// Mitsubishi GX Works2 project: 15속도제어   PLC: Q03UDV

PROGRAM MAIN
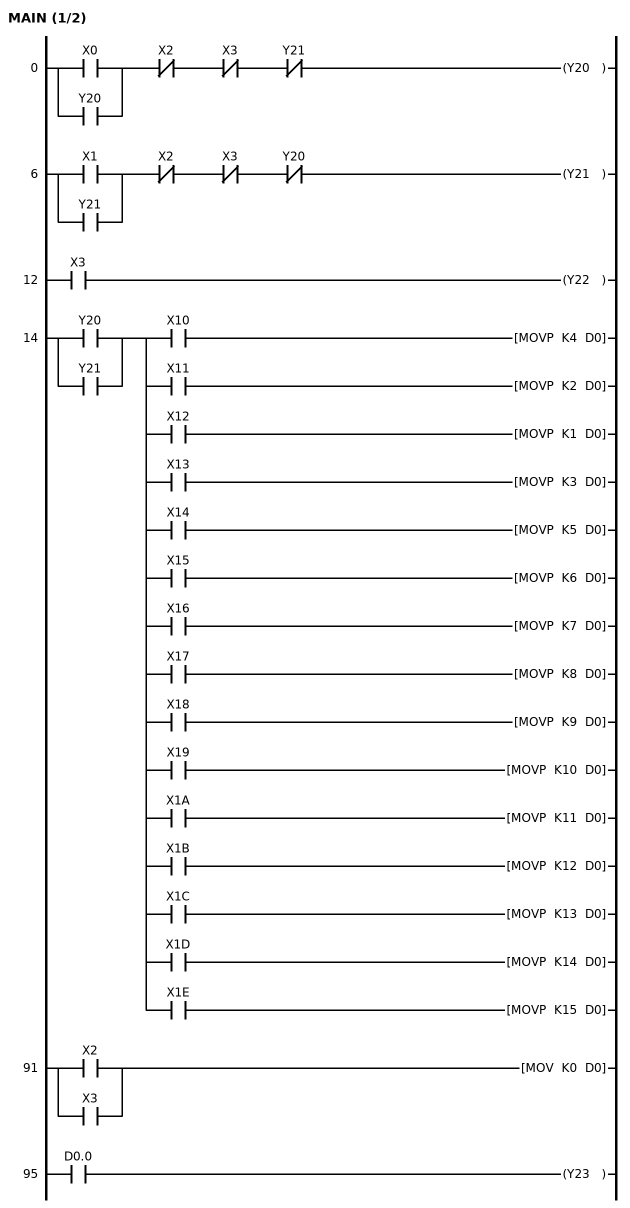
0     LD      X0
      OR      Y20
      ANI     X2
      ANI     X3
      ANI     Y21
      OUT     Y20
6     LD      X1
      OR      Y21
      ANI     X2
      ANI     X3
      ANI     Y20
      OUT     Y21
12    LD      X3
      OUT     Y22
14    LD      Y20
      OR      Y21
      MPS
      AND     X10
      MOVP    K4 D0
      MRD
      AND     X11
      MOVP    K2 D0
      MRD
      AND     X12
      MOVP    K1 D0
      MRD
      AND     X13
      MOVP    K3 D0
      MRD
      AND     X14
      MOVP    K5 D0
      MRD
      AND     X15
      MOVP    K6 D0
      MRD
      AND     X16
      MOVP    K7 D0
      MRD
      AND     X17
      MOVP    K8 D0
      MRD
      AND     X18
      MOVP    K9 D0
      MRD
      AND     X19
      MOVP    K10 D0
      MRD
      AND     X1A
      MOVP    K11 D0
      MRD
      AND     X1B
      MOVP    K12 D0
      MRD
      AND     X1C
      MOVP    K13 D0
      MRD
      AND     X1D
      MOVP    K14 D0
      MPP
      AND     X1E
      MOVP    K15 D0
91    LD      X2
      OR      X3
      MOV     K0 D0
95    LD      D0.0
      OUT     Y23
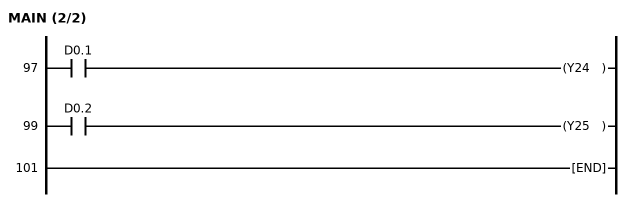
97    LD      D0.1
      OUT     Y24
99    LD      D0.2
      OUT     Y25
101   END
END_PROGRAM
